GLOBALCONSTANTS ResetButtonDiagCodes (* PLCopen Safety Part 1 Ch. 6.1.6 - SF_ResetButton-specific DiagCode values *)
  (* Standard: 61499-1; Description: Copyright (c) 2026 Meisterschulen am Ostbahnhof This program and the accompanying materials are made available under the terms of the Eclipse Public License 2.0 which is available at https://www.eclipse.org/legal/epl-2.0/ SPDX-License-Identifier: EPL-2.0 *)
  (* Version 1.0, 2026-10-09, Franz Höpfinger, Meisterschulen am Ostbahnhof, Source: PLCopen TC5 Safety Part 1, Version 2.10, Chapter 6.1.6 DiagCode table. See also DiagCodes.gcf for the shared IDLE code. *)
  PACKAGE logiBUS::safety::PLCopen::const;
  VAR_GLOBAL CONSTANT
    WAIT_R_TRIG : WORD := 16#83E2; (* 83E2 - enabled, waiting for rising edge on ResetIn *)
    WAIT_F_TRIG : WORD := 16#83F2; (* 83F2 - ResetIn is TRUE, waiting for falling edge *)
    RESET_DETECTED : WORD := 16#8000; (* 8000 - valid trailing-edge reset, 1-cycle pulse *)
    PARAMETER_ERROR : WORD := 16#C000; (* C000 - TrailingMinimum > TrailingMaximum OR TrailingMinimum < 100ms *)
    RESET_ERROR : WORD := 16#C001; (* C001 - ResetIn was already TRUE when ResetRequested became TRUE *)
    ERROR_TRAILING_MAXIMUM : WORD := 16#C3E0; (* C3E0 - TrailingMaximum elapsed before F_TRIG. Waiting for R_TRIG *)
    ERROR_TRAILING_MINIMUM : WORD := 16#C3F0; (* C3F0 - F_TRIG before TrailingMinimum elapsed. Waiting for R_TRIG *)
  END_VAR
END_GLOBALCONSTANTS
